(* PLC project TestProject.project, iec-st-tools CODESYS CODESYS V3.5 SP19 Patch 6 *)
(* stored: creationDateTime 2026-02-26T16:23:28.3873371, modificationDateTime 2026-02-26T16:23:28.3873371 *)

TYPE TestStruct : STRUCT
  Value : INT := 0;
  IsValid : BOOL := FALSE;
  Name : STRING := '';
END_STRUCT;
END_TYPE

TYPE TestEnum : (stIdle, stactive, stError);
END_TYPE

VAR_GLOBAL  (* Globals *)
  G_SafeInvertTest : INT := 0;
END_VAR

FUNCTION SafeInvert
  VAR_INPUT
    value : INT;
  END_VAR

            IF value = -32768 THEN
    SafeInvert := 32767;
ELSE
    SafeInvert := 0 - value;
END_IF;

          
END_FUNCTION
